TYPE TcoDatamanAcquisitionStatus_v_5_x_x : STRUCT
    TriggerReady AT %I* : BOOL;
    TriggerAcknowledge AT %I* : BOOL;
    Acquiring AT %I* : BOOL;
    MissedAcquisition AT %I* : BOOL;
    TriggerID AT %I* : UINT;
END_STRUCT
END_TYPE

(* stored: Version 1.1.0.1, ProductVersion 3.1.4024.11
   DUT TcoDatamanAcquisitionStatus_v_5_x_x: Id {14df66c4-970c-49dc-99e6-84ac8732a883} *)
